FUNCTION_BLOCK E_SR_SYM (* Event-driven bistable, symmetric Start-Up Behaviour *)
  (* Standard: 61499-1 Annex A; Description: Copyright (c) 2017 fortiss GmbH, HR Agrartechnik GmbH This program and the accompanying materials are made available under the terms of the Eclipse Public License 2.0 which is available at https://www.eclipse.org/legal/epl-2.0/ SPDX-License-Identifier: EPL-2.0 *)
  (* Version 1.0, 2026-05-12, Franz Höpfinger, HR Agrartechnik GmbH, initial API and implementation and/or initial documentation *)
  PACKAGE iec61499::events;
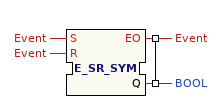
  EVENT_INPUT
    S; (* Set output Q *)
    R; (* Reset output Q *)
  END_EVENT
  EVENT_OUTPUT
    EO WITH Q; (* Output Q has changed *)
  END_EVENT
  VAR_OUTPUT
    Q : BOOL; (* value of flip flop *)
  END_VAR
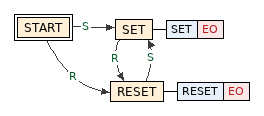
  EC_STATES
    START; (* Initial State *)
    SET : SET -> EO;
    RESET : RESET -> EO;
  END_STATES
  EC_TRANSITIONS
    START TO SET := S;
    SET TO RESET := R;
    RESET TO SET := S;
    START TO RESET := R;
  END_TRANSITIONS
  ALGORITHM SET IN ST: (* SET algorithm *)
Q := TRUE;
  END_ALGORITHM
  ALGORITHM RESET IN ST: (* RESET algorithm *)
Q := FALSE;
  END_ALGORITHM
END_FUNCTION_BLOCK
